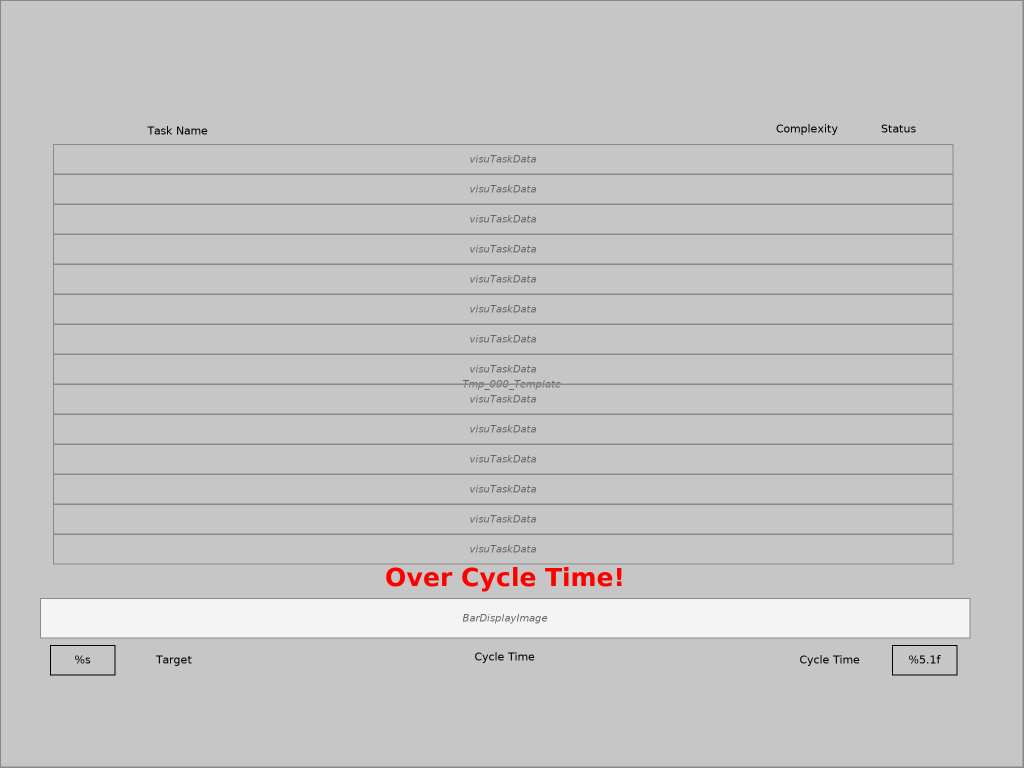
VISUALIZATION Prc_501_Cycle  // 1024x768
    Frame (0,0 1024x768)
        shows Tmp_000_Template(header := gHMIData.hmiHeader)
    BarDisplayImage (40,598 930x40), value: Mc_Global.part.CycleTimeActual, style: BarDisplayImage-Gray, scale format: %.1f, scale 0..100
    Label (40,642 930x30), "Cycle Time"
    Label (40,562 930x30), "Over Cycle Time!", invisible if: NOT Mc_Global.part.OverCycleTime
    Frame (53,144 900x30)
        shows visuTaskData(d := Mc_Global.part.tasks[1])
    Rectangle (892,645 65x30), "%5.1f", text variable: Mc_Global.part.CycleTimeActual
    Label (771,645 118x30), "Cycle Time"
    Rectangle (50,645 65x30), "%s", text variable: Mc_Global.part.CycleTimeTarget
    Label (115,645 118x30), "Target"
    Frame (53,174 900x30)
        shows visuTaskData(d := Mc_Global.part.tasks[2])
    Frame (53,204 900x30)
        shows visuTaskData(d := Mc_Global.part.tasks[3])
    Frame (53,234 900x30)
        shows visuTaskData(d := Mc_Global.part.tasks[4])
    Frame (53,264 900x30)
        shows visuTaskData(d := Mc_Global.part.tasks[5])
    Frame (53,294 900x30)
        shows visuTaskData(d := Mc_Global.part.tasks[6])
    Frame (53,324 900x30)
        shows visuTaskData(d := Mc_Global.part.tasks[7])
    Frame (53,354 900x30)
        shows visuTaskData(d := Mc_Global.part.tasks[8])
    Frame (53,384 900x30)
        shows visuTaskData(d := Mc_Global.part.tasks[9])
    Frame (53,414 900x30)
        shows visuTaskData(d := Mc_Global.part.tasks[10])
    Frame (53,444 900x30)
        shows visuTaskData(d := Mc_Global.part.tasks[11])
    Frame (53,474 900x30)
        shows visuTaskData(d := Mc_Global.part.tasks[12])
    Frame (53,504 900x30)
        shows visuTaskData(d := Mc_Global.part.tasks[13])
    Frame (53,534 900x30)
        shows visuTaskData(d := Mc_Global.part.tasks[14])
    Label (103,116 150x30), "Task Name"
    Label (776,114 62x30), "Complexity"
    Label (844,114 109x30), "Status"
END_VISUALIZATION

(* stored: Version 1.1.0.1, ProductVersion 3.1.4024.12
   Visu Prc_501_Cycle: Id {be3e1f29-3c27-4c3e-8e90-a74c740438d6} *)
